FUNCTION_BLOCK FB_Breeder EXTENDS FB_Station
VAR
	iBreedableArr			: ARRAY [1..50] OF INT;
	iLastBreedIndex			: INT;
END_VAR

METHOD Breeding : INT
VAR
	stTempUnit				: ST_Unit;
	iTempIndex				: INT;
	iBreedIndex				: INT;
	iBreedCounter			: INT;
END_VAR
Breeding := 0;
IF iLastIndex > 1 THEN
	FOR iTempIndex := 1 TO iLastIndex BY 1 DO
		stTempUnit := stUnitArr[iTempIndex];
		IF stTempUnit.iProgress < 6 THEN
			stTempUnit.iProgress := stTempUnit.iProgress + 1;
			stUnitArr[iTempIndex] := stTempUnit;
		ELSE
			iBreedIndex := iBreedIndex + 1;
			iBreedableArr[iBreedIndex] := iTempIndex;
			iLastBreedIndex := iBreedIndex;
		END_IF
	END_FOR
END_IF

IF iLastBreedIndex > 1 THEN
	FOR iBreedIndex := 1 TO iLastBreedIndex BY 1 DO
		stTempUnit := stUnitArr[iBreedableArr[iBreedIndex]];
		stTempUnit.iProgress := 0;
		stUnitArr[iBreedableArr[iBreedIndex]] := stTempUnit;
		iBreedCounter := iBreedCounter + 1;
	END_FOR
	iLastBreedIndex := 0;
	Breeding := iBreedCounter / 2;
END_IF
END_METHOD

END_FUNCTION_BLOCK

(* stored: Version 1.1.0.1, ProductVersion 3.1.4024.12
   POU FB_Breeder: Id {f42eb3d6-1236-45b8-ba11-23c59e597994}, SpecialFunc None
   Method Breeding: Id {e3a38cc5-d3c4-4a1d-8c2b-e478c877839a} *)
